// Mitsubishi GX Works2 project: q07   PLC: Q02/Q02H

PROGRAM MAIN
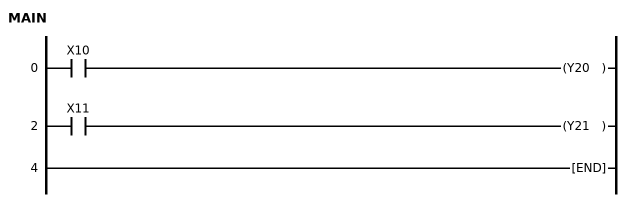
0     LD      X10
      OUT     Y20
2     LD      X11
      OUT     Y21
4     END
END_PROGRAM

PROGRAM touth
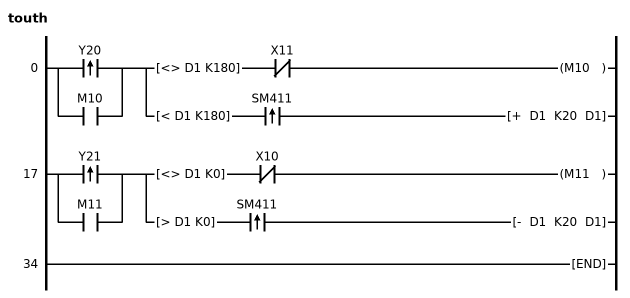
0     LDP     Y20
      OR      M10
      MPS
      AND<>   D1 K180
      ANI     X11
      OUT     M10
      MPP
      AND<    D1 K180
      ANDP    SM411
      +       D1 K20 D1
17    LDP     Y21
      OR      M11
      MPS
      AND<>   D1 K0
      ANI     X10
      OUT     M11
      MPP
      AND>    D1 K0
      ANDP    SM411
      -       D1 K20 D1
34    END
END_PROGRAM

PROGRAM ALARM
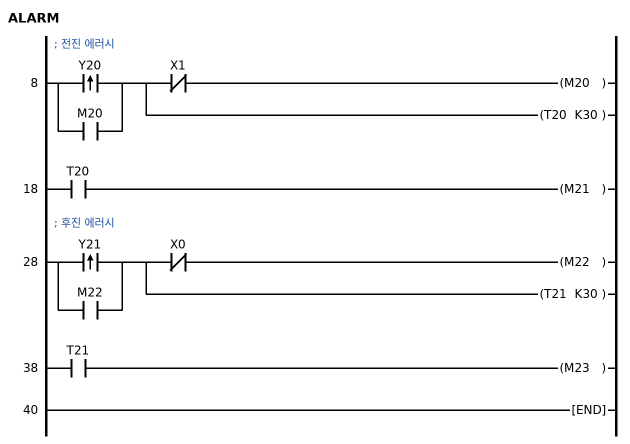
; 전진 에러시
8     LDP     Y20
      OR      M20
      MPS
      ANI     X1
      OUT     M20
      MPP
      OUT     T20 K30
18    LD      T20
      OUT     M21
; 후진 에러시
28    LDP     Y21
      OR      M22
      MPS
      ANI     X0
      OUT     M22
      MPP
      OUT     T21 K30
38    LD      T21
      OUT     M23
40    END
END_PROGRAM
